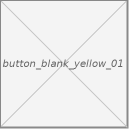
VISUALIZATION Yellow_Ind  // 129x129
VAR_IN_OUT
	m_Input_Inst : None;
END_VAR
    Image (0,0 127x127), invisible if: (m_Input_Inst) <> 0, image: button_blank_gray_01
    Image (0,0 127x127), invisible if: (NOT m_Input_Inst) <> 0, image: button_blank_yellow_01
END_VISUALIZATION

(* stored: Version 1.1.0.1, ProductVersion 3.1.4018.2
   Visu Yellow_Ind: Id {04181acb-3658-4b4f-b878-8179c2b213a4} *)
